PROGRAM StateMachine
VAR
	bPizzaOnDeck : BOOL;
	bPizzaInOven : BOOL;
	bPizzaDone	 : BOOL;
	
	//timers
	fbMyTimer	 : TON;
	
	bLoadPIzza	: BOOL; // put pizza on input side
	bRemovepizza: BOOL;	//remove pizza off output side
	
	iState 		: DINT;
	sStateDesc	: STRING;
	
	//trigs
	fbMyTrigger_RTRIG	: R_TRIG; //pizza counter
	
	bBuzzer		: BOOL;
	bLight		: BOOL;
	
	iTotalPizzasCooked	: UDINT;

	condition: BOOL;
END_VAR


//youtube "Learning PLC with ST EP7 - State Machines



IF bPizzaOnDeck AND NOT bPizzaInOven THEN
	bPizzaOnDeck	:= FALSE;
	bPizzaInOven 	:= TRUE;
END_IF

IF bLoadPIzza THEN
	bLoadPizza		:= FALSE;
	bPizzaOnDeck	:= TRUE;
END_IF

IF bRemovePizza THEN
	bPizzaDone		:= FALSE;
	bPizzaOnDeck	:= FALSE;
END_IF

CASE iState OF

	0:	// Wait for pizza in oven
		sStateDesc := 'Waiting on that pizza';
		IF bPizzaInOven THEN		
			iState := 10; //move on
		END_IF
	10: //We just got a pizza!
		sStateDesc := 'Baking that pizza-boi';
		fbMyTimer(IN:=TRUE,PT:=T#3S);
		IF fbMyTimer.Q THEN
			fbMyTimer(IN:=FALSE);
			iState := 20;
		END_IF
		
	20: // Can we move the pizza out? Its going to burn else
	
		IF NOT bPizzaDone THEN
			//simulate conveyor
			bPizzaInOven 	:= FALSE;
			bPizzaDone 		:= TRUE;
			bBuzzer			:= FALSE;

			iState 			:= 30;

		ELSE
			bBuzzer := TRUE;
		END_IF
	
	30: //Pizzas just removed. On output tray
		iTotalPizzasCooked 	:= iTotalPizzasCooked +1;
		iState 				:= 0;  // Go wait for new pizza
	
ELSE
	sStateDesc := 'Invalid state'
;
	
	;
END_CASE



fbMyTimer(IN:=bPizzaInOven,PT:=T#3S);

bBuzzer := fbMyTimer.Q;

fbMyTrigger_RTRIG(clk:=fbMyTimer.Q);

IF fbMyTrigger_RTRIG.Q THEN
	iTotalPizzasCooked := iTotalPizzasCooked +1;
END_IF

END_PROGRAM

(* stored: Version 1.1.0.1, ProductVersion 3.1.4024.10
   POU StateMachine: Id {963f2670-b1fa-404a-9599-e89587cf9076}, SpecialFunc None *)
